Omron CX-Programmer project NewProject (CX-Programmer 9.45)

# PLC NewPLC1: CP1H XA

## Global symbols (name address type ; comment)
W0.07 BOOL  ; ACCELERATION START
BUTTON_1 2.04 BOOL
BUTTON_1_UP 1.07 BOOL
BUTTON_2 2.03 BOOL
BUTTON_2_DOWN 1.06 BOOL
BUTTON_2_UP 1.05 BOOL
BUTTON_3 2.02 BOOL
BUTTON_3_DOWN 1.04 BOOL
BUTTON_3_UP 1.03 BOOL
BUTTON_4 2.01 BOOL
BUTTON_4_DOWN 1.02 BOOL
BUTTON_4_UP 1.01 BOOL
BUTTON_5 2.00 BOOL
BUTTON_5_DOWN 1.00 BOOL
BUTTON_OPEN 2.05 BOOL
BUTTON_OPEN_LAMP 103.05 BOOL
BUTTON_SHUT 2.06 BOOL
BUTTON_SHUT_LAMP 103.06 BOOL
DOOR_OPEN 100.00 BOOL
DOOR_SHUT 100.01 BOOL
LIMIT_1 0.10 BOOL
LIMIT_2 0.07 BOOL
LIMIT_3 0.06 BOOL
LIMIT_4 0.05 BOOL
LIMIT_5 0.04 BOOL
LIMIT_OPEN 0.01 BOOL
LIMIT_SHUT 0.00 BOOL
WINCH_MOTOR 210 WORD
_HOLD_VALUE 2921 NUMBER

## Program NewProgram1 (cyclic task 0)
Local symbols
CurrentState W10 INT
DESTINATION D925 DINT
FIVE_DOWN W8.07 BOOL
FIVE_INT W8.12 BOOL
FOUR_DOWN W8.05 BOOL
FOUR_INT W8.11 BOOL
FOUR_UP W8.06 BOOL
FunkyState W40 INT
InitState D101 INT
MovingState D102 INT
ONE_INT W8.08 BOOL
ONE_UP W8.00 BOOL
SAFE_TO_OPEN D103 INT
START_BIT W1.02 BOOL
THREE_DOWN W8.03 BOOL
THREE_INT W8.10 BOOL
THREE_UP W8.04 BOOL
TRIGGER_2 W99.01 BOOL
TWO_DOWN W8.01 BOOL
TWO_INT W8.09 BOOL
TWO_UP W8.02 BOOL
_FLOOR_1_POS D960 DINT
_FLOOR_2_POS D945 DINT
_FLOOR_3_POS D940 DINT
_FLOOR_4_POS D935 DINT
_FLOOR_5_POS D930 DINT
temphold D60 DINT

### Section Section1

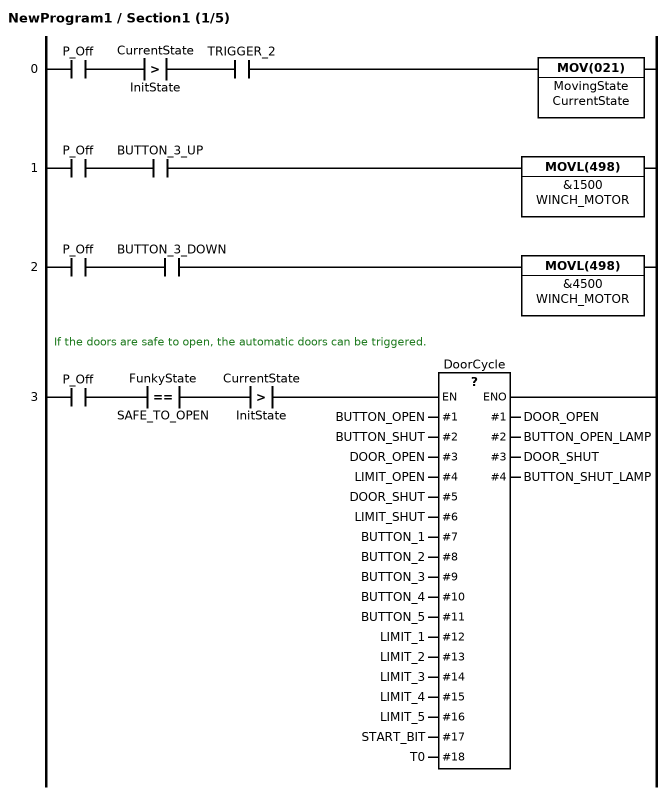
; rung 0
LD P_Off
AND>(320) CurrentState InitState
AND TRIGGER_2
MOV(021) MovingState CurrentState
; rung 1
LD P_Off
AND BUTTON_3_UP
MOVL(498) &1500 WINCH_MOTOR
; rung 2
LD P_Off
AND BUTTON_3_DOWN
MOVL(498) &4500 WINCH_MOTOR
; rung 3: If the doors are safe to open, the automatic doors can be triggered.
LD P_Off
AND=(300) FunkyState SAFE_TO_OPEN
AND>(320) CurrentState InitState
CALL DoorCycle : ? (#1 := BUTTON_OPEN, #2 := BUTTON_SHUT, #3 := DOOR_OPEN, #4 := LIMIT_OPEN, #5 := DOOR_SHUT, #6 := LIMIT_SHUT, #7 := BUTTON_1, #8 := BUTTON_2, #9 := BUTTON_3, #10 := BUTTON_4, #11 := BUTTON_5, #12 := LIMIT_1, #13 := LIMIT_2, #14 := LIMIT_3, #15 := LIMIT_4, #16 := LIMIT_5, #17 := START_BIT, #18 := T0)

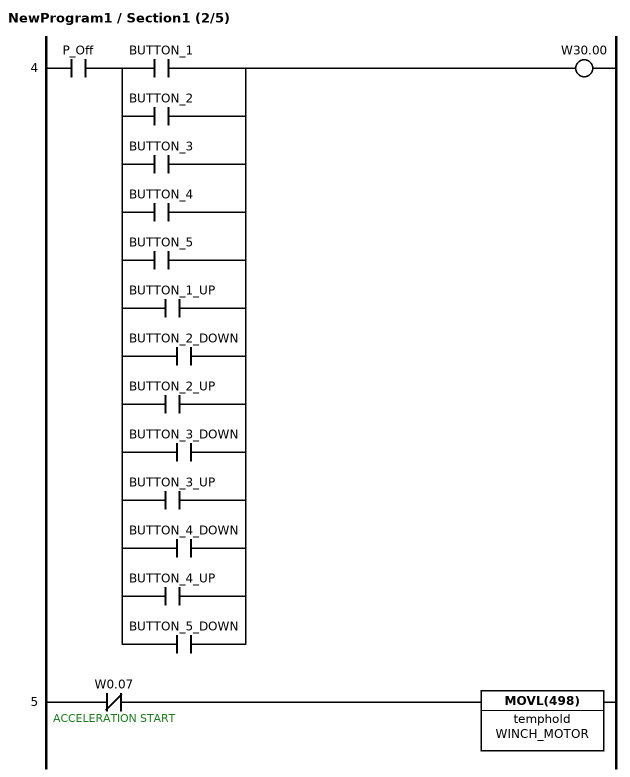
; rung 4
LD P_Off
LD BUTTON_1
OR BUTTON_2
OR BUTTON_3
OR BUTTON_4
OR BUTTON_5
OR BUTTON_1_UP
OR BUTTON_2_DOWN
OR BUTTON_2_UP
OR BUTTON_3_DOWN
OR BUTTON_3_UP
OR BUTTON_4_DOWN
OR BUTTON_4_UP
OR BUTTON_5_DOWN
ANDLD
OUT W30.00
; rung 5
LDNOT W0.07  ; ACCELERATION START
MOVL(498) temphold WINCH_MOTOR

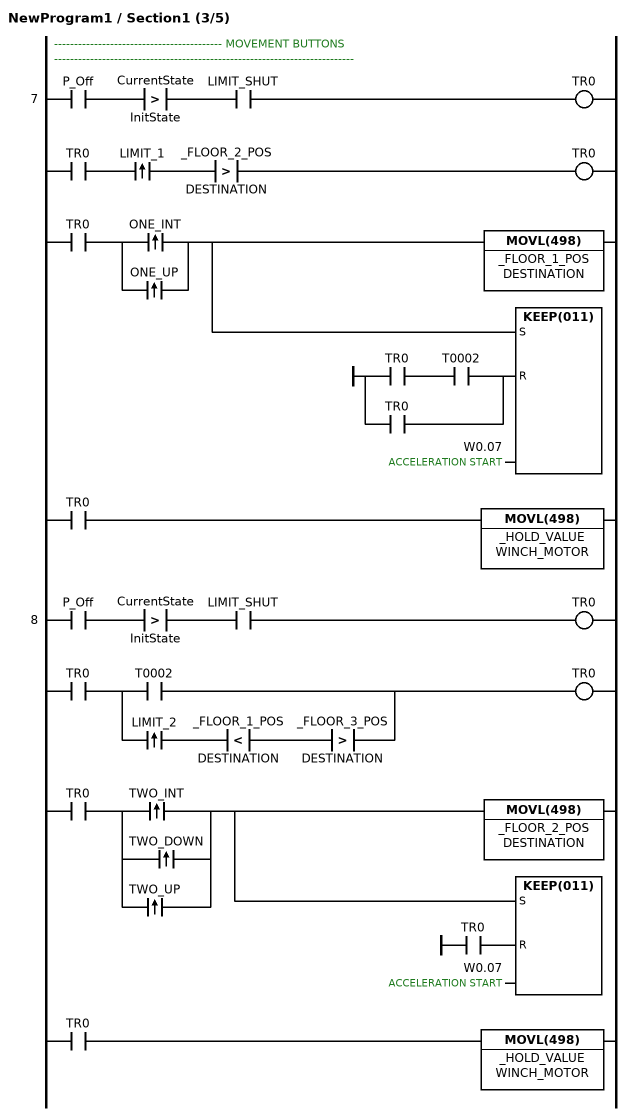
; rung 7: ------------------------------------------ MOVEMENT BUTTONS ---------------------------------------------------------------------------
LD P_Off
AND>(320) CurrentState InitState
AND LIMIT_SHUT
OUT TR0
@LD ONE_INT
@OR ONE_UP
ANDLD
MOVL(498) _FLOOR_1_POS DESTINATION
LD TR0
AND T0002
LD TR0
@AND LIMIT_1
AND>L(321) _FLOOR_2_POS DESTINATION
OUT TR0
ORLD
KEEP(011) W0.07  ; ACCELERATION START
LD TR0
MOVL(498) _HOLD_VALUE WINCH_MOTOR
; rung 8
LD P_Off
AND>(320) CurrentState InitState
AND LIMIT_SHUT
OUT TR0
@LD TWO_INT
@OR TWO_DOWN
@OR TWO_UP
ANDLD
MOVL(498) _FLOOR_2_POS DESTINATION
LD TR0
LD T0002
@LD LIMIT_2
AND<L(311) _FLOOR_1_POS DESTINATION
AND>L(321) _FLOOR_3_POS DESTINATION
ORLD
ANDLD
OUT TR0
KEEP(011) W0.07  ; ACCELERATION START
LD TR0
MOVL(498) _HOLD_VALUE WINCH_MOTOR

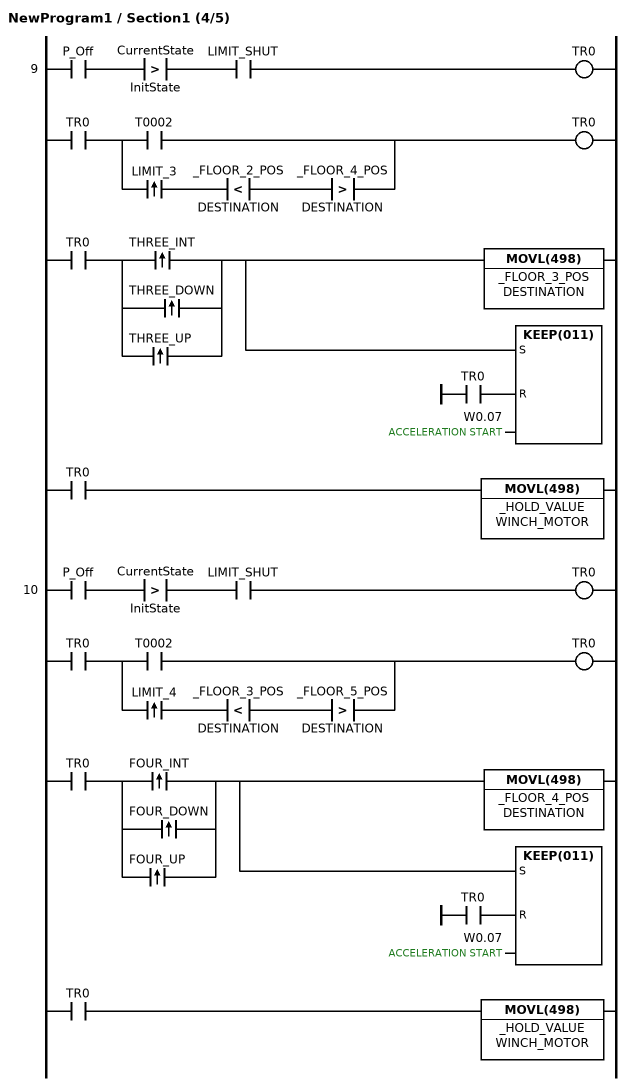
; rung 9
LD P_Off
AND>(320) CurrentState InitState
AND LIMIT_SHUT
OUT TR0
@LD THREE_INT
@OR THREE_DOWN
@OR THREE_UP
ANDLD
MOVL(498) _FLOOR_3_POS DESTINATION
LD TR0
LD T0002
@LD LIMIT_3
AND<L(311) _FLOOR_2_POS DESTINATION
AND>L(321) _FLOOR_4_POS DESTINATION
ORLD
ANDLD
OUT TR0
KEEP(011) W0.07  ; ACCELERATION START
LD TR0
MOVL(498) _HOLD_VALUE WINCH_MOTOR
; rung 10
LD P_Off
AND>(320) CurrentState InitState
AND LIMIT_SHUT
OUT TR0
@LD FOUR_INT
@OR FOUR_DOWN
@OR FOUR_UP
ANDLD
MOVL(498) _FLOOR_4_POS DESTINATION
LD TR0
LD T0002
@LD LIMIT_4
AND<L(311) _FLOOR_3_POS DESTINATION
AND>L(321) _FLOOR_5_POS DESTINATION
ORLD
ANDLD
OUT TR0
KEEP(011) W0.07  ; ACCELERATION START
LD TR0
MOVL(498) _HOLD_VALUE WINCH_MOTOR

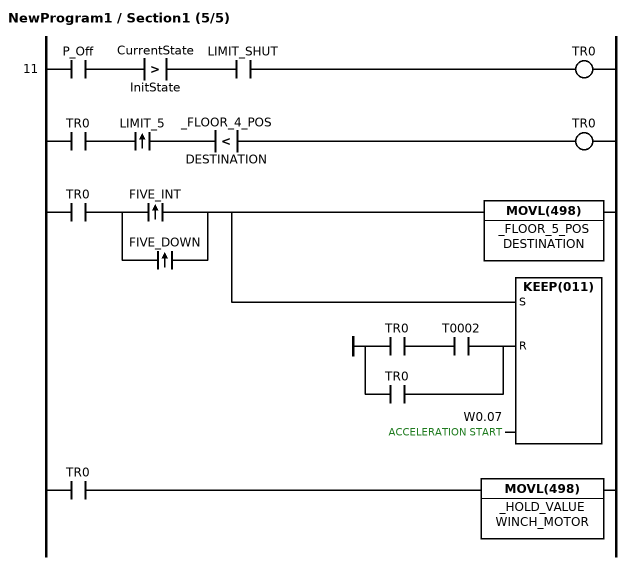
; rung 11
LD P_Off
AND>(320) CurrentState InitState
AND LIMIT_SHUT
OUT TR0
@LD FIVE_INT
@OR FIVE_DOWN
ANDLD
MOVL(498) _FLOOR_5_POS DESTINATION
LD TR0
AND T0002
LD TR0
@AND LIMIT_5
AND<L(311) _FLOOR_4_POS DESTINATION
OUT TR0
ORLD
KEEP(011) W0.07  ; ACCELERATION START
LD TR0
MOVL(498) _HOLD_VALUE WINCH_MOTOR

### Section END
; rung 0
END(001)